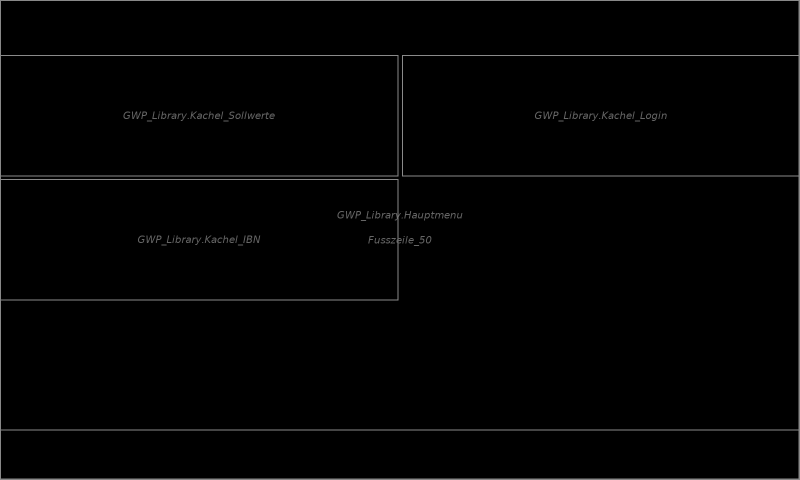
VISUALIZATION Hauptmenu  // 800x480
    Frame (0,0 800x430)
        shows GWP_Library.Hauptmenu()
    Frame (0,179 398x121)
        shows GWP_Library.Kachel_IBN()
        OnMouseClick: change screen: IBS_Menu
    Frame (0,55 398x121)
        shows GWP_Library.Kachel_Sollwerte()
        OnMouseClick: change screen: Sollwertmenu
    Frame (402,55 398x121)
        shows GWP_Library.Kachel_Login()
        OnMouseClick: change screen: Login
    Frame (0,0 800x480)
        shows Fusszeile_50()
END_VISUALIZATION

(* stored: Version 1.1.0.1, ProductVersion 3.1.4022.6
   Visu Hauptmenu: Id {ea5afc57-6b3b-4d29-9a02-2714784943e5} *)
